{attribute 'GeneratedUsingTerminal: EL3423-0000-0017'}
{attribute addProperty BoxType "EL3423-0000-0017"}
{attribute addProperty Id "Reset_IntervalAT %Q*BOOL1"}
{attribute addProperty CRC "360233940"}
{attribute addProperty Size "1"}
TYPE Total_Interval_1578BBD4 :
STRUCT
	{attribute addProperty Name "Reset_Interval"}
	Reset_Interval AT %Q* : BOOL;
END_STRUCT
END_TYPE

(* stored: Version 1.2.0.0, ProductVersion 3.1.4024.9
   DUT Total_Interval_1578BBD4: Id {0f6e16fc-59d1-4e08-b62e-a2cdd8df9032} *)
